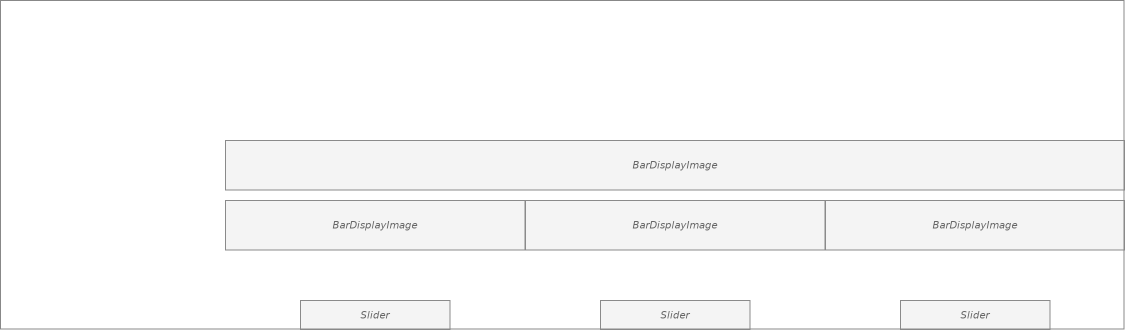
VISUALIZATION Visualization  // 1125x330
    Slider (600,300 150x30), variable: MAIN.Vat2, scale 0..3000
    Slider (900,300 150x30), variable: MAIN.Vat3, scale 0..5000
    Slider (300,300 150x30), variable: MAIN.Vat1, scale 0..2000
    BarDisplayImage (225,200 300x50), value: MAIN.Vat1, style: BarDisplayImage-Gray, scale format: %.1f, scale 0..2000
    BarDisplayImage (525,200 300x50), value: MAIN.Vat2, style: BarDisplayImage-Gray, scale format: %.1f, scale 0..3000
    BarDisplayImage (825,200 300x50), value: MAIN.Vat3, style: BarDisplayImage-Gray, scale format: %.1f, scale 0..5000
    BarDisplayImage (225,140 900x50), value: MAIN.TotalOutput, style: BarDisplayImage-Gray, scale format: %.1f, scale 0..10000
END_VISUALIZATION

(* stored: Version 1.1.0.1, ProductVersion 3.1.4024.12
   Visu Visualization: Id {2056f3c0-6c6b-4927-b55f-bc3e8f5efd62} *)
